PROGRAM simIniciaProg_Manual_3
VAR
	bSimIniciaProg: BOOL:= FALSE;
	posicaoAtual: STRING;
	envialog: STRING;
	bGravarConfigPosicao_Reator: BOOL;
END_VAR


gvl_p.arrStatusEstufas[gvl.actEst].startManual := TRUE;

bGravarConfigPosicao_Reator:= TRUE;

END_PROGRAM

(* stored: Version 1.1.0.1, ProductVersion 3.1.4024.12
   POU simIniciaProg_Manual_3: Id {c04a003d-5cbb-4366-a4db-04ad738f5bc9}, SpecialFunc None *)
